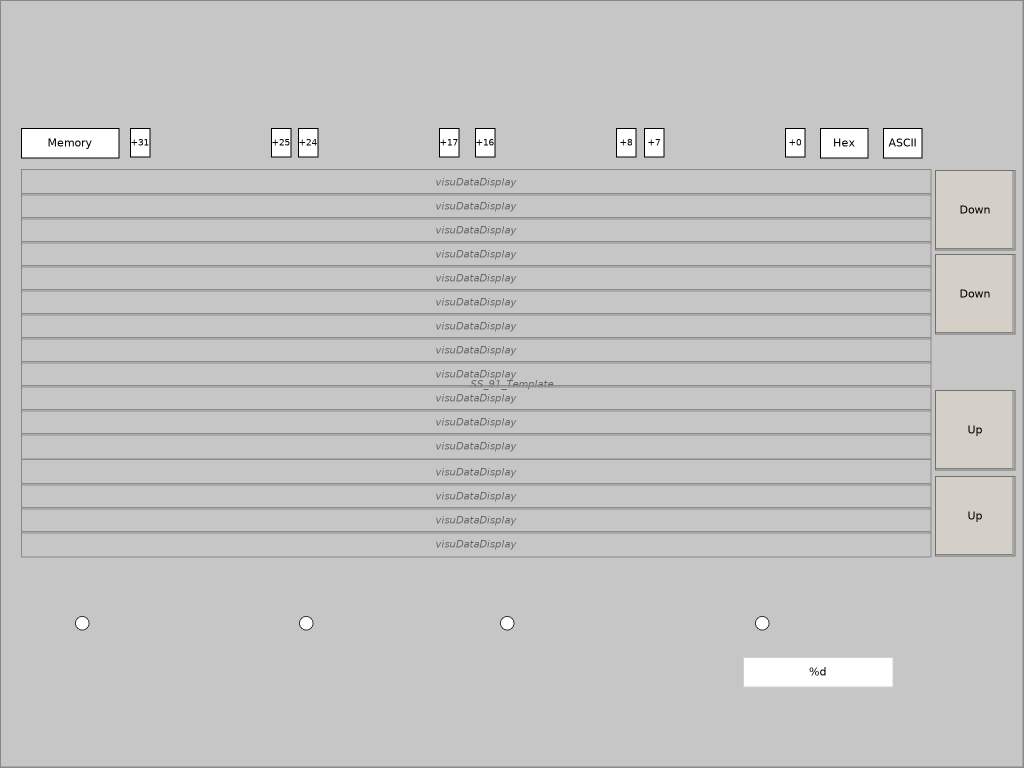
VISUALIZATION SS_99_DataDisplay  // 1024x768
    Frame (0,0 1024x768)
        shows SS_91_Template(header := HMIData.hmiHeader)
    Frame (21,169 910x26)
        shows visuDataDisplay(d := ioView.row01)
    Frame (21,193 910x26)
        shows visuDataDisplay(d := ioView.row02)
    Frame (21,217 910x26)
        shows visuDataDisplay(d := ioView.row03)
    Frame (21,241 910x26)
        shows visuDataDisplay(d := ioView.row04)
    Frame (21,265 910x26)
        shows visuDataDisplay(d := ioView.row05)
    Frame (21,289 910x26)
        shows visuDataDisplay(d := ioView.row06)
    Frame (21,313 910x26)
        shows visuDataDisplay(d := ioView.row07)
    Frame (21,337 910x26)
        shows visuDataDisplay(d := ioView.row08)
    Frame (21,361 910x26)
        shows visuDataDisplay(d := ioView.row09)
    Frame (21,385 910x26)
        shows visuDataDisplay(d := ioView.row10)
    Frame (21,409 910x26)
        shows visuDataDisplay(d := ioView.row11)
    Frame (21,433 910x26)
        shows visuDataDisplay(d := ioView.row12)
    Rectangle (21,128 98x30), "Memory"
    Rectangle (883,128 39x30), "ASCII"
    Rectangle (820,128 48x30), "Hex"
    Rectangle (785,128 20x29), "+0"
    Rectangle (644,128 20x29), "+7"
    Rectangle (475,128 20x29), "+16"
    Rectangle (616,128 20x29), "+8"
    Rectangle (439,128 20x29), "+17"
    Rectangle (298,128 20x29), "+24"
    Rectangle (271,128 20x29), "+25"
    Rectangle (130,128 20x29), "+31"
    Frame (21,459 910x26)
        shows visuDataDisplay(d := ioView.row13)
    Frame (21,483 910x26)
        shows visuDataDisplay(d := ioView.row14)
    Frame (21,507 910x26)
        shows visuDataDisplay(d := ioView.row15)
    Frame (21,531 910x26)
        shows visuDataDisplay(d := ioView.row16)
    Button (935,476 80x80), "Up"
        tap ioView.btnRaiseFaster
    Button (935,390 80x80), "Up"
        tap ioView.btnRaise
    Button (935,254 80x80), "Down"
        tap ioView.btnLower
    Button (935,170 80x80), "Down"
        tap ioView.btnLowerFaster
    RadioButton (753,583 150x80), variable: ioView.memtype
    RadioButton (73,583 150x80), variable: ioView.memsize
    RadioButton (297,583 230x80), variable: ioView.memHexDisplay
        p340057476: HEX/DEC
    RadioButton (498,583 235x80), variable: ioView.memswap
        p2481256679: SIEMENS/754
    Textfield (743,657 150x30), "%d", text variable: ioView.memoffset
        OnMouseClick: write ioView.memoffset via VisuDialogs.Numpad
END_VISUALIZATION

(* stored: Version 1.1.0.1, ProductVersion 3.1.4024.12
   Visu SS_99_DataDisplay: Id {81d00564-ef7e-46db-b7df-86ab8833ec42} *)
